// Convert nCurrGantry to um (smaller number) to read out in epics
M2L0.fCurrGantryY_um := LINT_TO_REAL(M2L0.nCurrGantryY) / 1000;
M2L0.fCurrGantryX_um := LINT_TO_REAL(M2L0.nCurrGantryX) / 1000;

// FB_MotionStage's for non-piezo axes
fbMotionStage_m7(stMotionStage:=M7);
fbMotionStage_m8(stMotionStage:=M8);
fbMotionStage_m9(stMotionStage:=M9);
fbMotionStage_m10(stMotionStage:=M10);
fbMotionStage_m11(stMotionStage:=M11);
fbMotionStage_m12(stMotionStage:=M12);

// Calculate RMS Error:
fbYRMSErrorM2L0(stMotionStage:=M7,
                fMaxRMSError=>fMaxYRMSErrorM2L0,
                fMinRMSError=>fMinYRMSErrorM2L0);

fbXRMSErrorM2L0(stMotionStage:=M9,
                fMaxRMSError=>fMaxXRMSErrorM2L0,
                fMinRMSError=>fMinXRMSErrorM2L0);

fbPitchRMSErrorM2L0(stMotionStage:=M11,
                fMaxRMSError=>fMaxPitchRMSErrorM2L0,
                fMinRMSError=>fMinPitchRMSErrorM2L0);

fbBenderRMSErrorM2L0(stMotionStage:=M12,
                fMaxRMSError=>fMaxBenderRMSErrorM2L0,
                fMinRMSError=>fMinBenderRMSErrorM2L0);

// Pitch Control
//fbM2L0PitchControl(Pitch:=GVL_M2L0.M2L0_Pitch,
                   //Stepper:=M11,
                   //lrCurrentSetpoint:=M11.fPosition,
                   //q_bDone=>bM2L0PitchDone,
                   //q_bBusy=>bM2L0PitchBusy);
// When STO hit, need to reset SP
//IF NOT M11.bHardwareEnable THEN
    //M11.fPosition := M11.stAxisStatus.fActPosition;
//END_IF

// Raw Encoder Counts For Epics
nEncCntYupM2L0 := ULINT_TO_UDINT(M2L0.fbRunHOMS.stYupEnc.Count);
nEncCntYdwnM2L0 := ULINT_TO_UDINT(M2L0.fbRunHOMS.stYdwnEnc.Count);
nEncCntXupM2L0 := ULINT_TO_UDINT(M2L0.fbRunHOMS.stXupEnc.Count);
nEncCntXdwnM2L0 := ULINT_TO_UDINT(M2L0.fbRunHOMS.stXdwnEnc.Count);
nEncCntPitchM2L0 := LINT_TO_UDINT(GVL_M2L0.M2L0_Pitch.diEncCnt);

// Encoder Reference Values For Epics
nEncRefYupM2L0 := ULINT_TO_UDINT(GVL_M2L0_Constants.nYUP_ENC_REF);
nEncRefYdwnM2L0 := ULINT_TO_UDINT(GVL_M2L0_Constants.nYDWN_ENC_REF);
nEncRefXupM2L0 := ULINT_TO_UDINT(GVL_M2L0_Constants.nXUP_ENC_REF);
nEncRefXdwnM2L0 := ULINT_TO_UDINT(GVL_M2L0_Constants.nXDWN_ENC_REF);
mcReadParameterPitchM2L0(Axis:=M11.Axis,
                         Enable:=TRUE,
                         ParameterNumber:=MC_AxisParameter.AxisEncoderOffset,
                         ReadMode:=READMODE_CYCLIC,
                         Value=>fEncRefPitchM2L0_urad);

nEncRefPitchM2L0 := LREAL_TO_UDINT(ABS(fEncRefPitchM2L0_urad) * fEncLeverArm_mm);

//Coatings States With PMPS
M7.bPowerSelf :=FALSE;


//SP1L0

// FB_MotionStage's for non-piezo axes
fbMotionStage_m13(stMotionStage:=M13);
fbMotionStage_m14(stMotionStage:=M14);
fbMotionStage_m15(stMotionStage:=M15);
fbMotionStage_m16(stMotionStage:=M16);
fbMotionStage_m17(stMotionStage:=M17);


M13.bHardwareEnable := bSTO AND bTH1_POTL AND bTH1_NOTL;
M14.bHardwareEnable := bSTO AND bTH2_POTL AND bTH2_NOTL;
M15.bHardwareEnable := bSTO AND bTX_POTL AND bTX_NOTL;
M16.bHardwareEnable := bSTO;
M17.bHardwareEnable := bSTO;


    //Turn on Fan by default
    bFanOn := TRUE;






P_CoatingProtections();


// Logging
fbLogHandler();

END_PROGRAM

// ---- POUs/P_CoatingProtections.TcPOU
PROGRAM P_CoatingProtections
VAR
        fbStripProtMR1L0 : FB_MirrorTwoCoatingProtection := (
            sDevName := 'MR1L0:HOMS',
            nUpperCoatingBoundary := 13300000,
            sUpperCoatingType := 'L0-B4C',
            nLowerCoatingBoundary := 11800000,
            sLowerCoatingType := 'L0-NICKEL');

        fbStripProtMR2L0 : FB_MirrorTwoCoatingProtection := (
            sDevName := 'MR2L0:HOMS',
            nUpperCoatingBoundary := 14300000,
            sUpperCoatingType := 'NICKEL',
            nLowerCoatingBoundary := 12800000,
            sLowerCoatingType := 'B4C');
END_VAR

fbStripProtMR1L0(
    FFO := GVL_PMPS.g_FastFaultOutput1,
    nCurrentEncoderCount := MAIN.nEncCntYupM1L0,
    neVRange := PMPS.PMPS_GVL.stCurrentBeamParameters.neVRange,
    bReadPmpsDb:= MOTION_GVL.fbStandardPMPSDB.bReadPmpsDb,
    bUsePmpsDb := TRUE,
   );

fbStripProtMR2L0(
    FFO := GVL_PMPS.g_FastFaultOutput1,
    nCurrentEncoderCount := MAIN.nEncCntYupM2L0,
    neVRange := PMPS.PMPS_GVL.stCurrentBeamParameters.neVRange,
    bReadPmpsDb:= MOTION_GVL.fbStandardPMPSDB.bReadPmpsDb,
    bUsePmpsDb := TRUE,
);

END_PROGRAM

// ---- POUs/PRG_1_PlcTask.TcPOU
PROGRAM PRG_1_PlcTask
VAR

END_VAR

PRG_MR1L0_HOMS();
PRG_MR2L0_HOMS();
PRG_SP1L0_DCCM();
PRG_PMPS();

END_PROGRAM

// ---- POUs/PRG_MR1L0_HOMS.TcPOU
PROGRAM PRG_MR1L0_HOMS
VAR
    {attribute 'pytmc' := 'pv: MR1L0:HOMS:COATING'}
    fbCoatingStates: FB_PositionStatePMPS2D;
    {attribute 'pytmc' := '
      pv: MR1L0:HOMS:COATING:STATE:SET
      io: io
    '}
    eStateSet: E_MR1L0_CoatingStates;
    {attribute 'pytmc' := '
      pv: MR1L0:HOMS:COATING:STATE:GET
      io: i
    '}
    eStateGet: E_MR1L0_CoatingStates;

    fbYSetup: FB_StateSetupHelper;

    fbPitchSetup: FB_StateSetupHelper;
    stDefaultPitch : ST_PositionState := (
        fDelta:=194.94,
        fVelocity:=100,
        fAccel:=390,
        fDecel:=390,
        bMoveOk:=TRUE,
        bValid:=TRUE,
        bUseRawCounts:=TRUE
    );
    astCoatingStatesY: ARRAY[1..GeneralConstants.MAX_STATES] OF ST_PositionState;
    astCoatingStatesPitch: ARRAY[1..GeneralConstants.MAX_STATES] OF ST_PositionState;

        // MR1L0 Flow Press Sensors
    {attribute 'TcLinkTo' := '.fbFlow_1.iRaw := TIIB[EL3054_M1L0_FWM_PRSM]^AI Standard Channel 1^Value;
                                 .fbFlow_2.iRaw := TIIB[EL3054_M1L0_FWM_PRSM]^AI Standard Channel 2^Value;
                              .fbPress_1.iRaw := TIIB[EL3054_M1L0_FWM_PRSM]^AI Standard Channel 3^Value
    '}
    {attribute 'pytmc' := '
        pv: MR1L0:HOMS
    '}
    fbCoolingPanel : FB_Axilon_Cooling_2f1p;
    {attribute 'TcLinkTo' := 'TIIB[EP2008-0001_M1M2_VCV]^Channel 1^Output'}
    {attribute 'pytmc' := '
        pv: MR1L0:HOMS:VCV
        io: io
        field: ZNAM OFF
        field: ONAM ON
    '}
    bActivateVarCoolMR1L0 AT %Q* : BOOL;
END_VAR

fbYSetup(stPositionState:=GVL_States.stDefaultY, bSetDefault:=TRUE);
fbPitchSetup(stPositionState:=stDefaultPitch, bSetDefault:=TRUE);

// MR1L0 B4C
fbYSetup(stPositionState:=astCoatingStatesY[E_MR1L0_CoatingStates.L0B4C],
    sName:='L0B4C',
    sPmpsState:='MR1L0:HOMS-L0-B4C',
    nEncoderCount:=21171800
);
fbPitchSetup(stPositionState:=astCoatingStatesPitch[E_MR1L0_CoatingStates.L0B4C],
    sName:='L0B4C',
    sPmpsState:='MR1L0:HOMS-L0-B4C',
    nEncoderCount:=8602330
);

// MR1L0 Ni
fbYSetup(stPositionState:=astCoatingStatesY[E_MR1L0_CoatingStates.L0Ni],
    sName:='L0Ni',
    sPmpsState:='MR1L0:HOMS-L0-NICKEL',
    nEncoderCount:=9171800
);
fbPitchSetup(stPositionState:=astCoatingStatesPitch[E_MR1L0_CoatingStates.L0Ni],
    sName:='L0Ni',
    sPmpsState:='MR1L0:HOMS-L0-NICKEL',
    nEncoderCount:=8602330
);

// MR1L0_L1 B4C
fbYSetup(stPositionState:=astCoatingStatesY[E_MR1L0_CoatingStates.L1B4C],
    bValid:=FALSE,
    sName:='L1B4C',
    sPmpsState:='MR1L0:HOMS-L1-B4C',
    nEncoderCount:=21171800
);
fbPitchSetup(stPositionState:=astCoatingStatesPitch[E_MR1L0_CoatingStates.L1B4C],
    bValid:=FALSE,
    sName:='L1B4C',
    sPmpsState:='MR1L0:HOMS-L1-B4C',
    nEncoderCount:=11116030,
    fDelta:=974.66
);

// MR1L0_L1 Ni
fbYSetup(stPositionState:=astCoatingStatesY[E_MR1L0_CoatingStates.L1Ni],
    bValid:=FALSE,
    sName:='L1Ni',
    sPmpsState:='MR1L0:HOMS-L1-NICKEL',
    nEncoderCount:=9171800
);
fbPitchSetup(stPositionState:=astCoatingStatesPitch[E_MR1L0_CoatingStates.L1Ni],
    bValid:=FALSE,
    sName:='L1Ni',
    sPmpsState:='MR1L0:HOMS-L1-NICKEL',
    nEncoderCount:=11116030,
    fDelta:=974.66
);

fbCoatingStates(
    stMotionStage1:=Main.M1,
    stMotionStage2:=Main.M5,
    astPositionState1:=astCoatingStatesY,
    astPositionState2:=astCoatingStatesPitch,
    eEnumSet:=eStateSet,
    eEnumGet:=eStateGet,
    fbFFHWO:=GVL_PMPS.g_FastFaultOutput1,
    fbArbiter:=GVL_PMPS.g_fbArbiter1,
    bEnableMotion:=TRUE,
    bEnableBeamParams:=TRUE,
    sDeviceName:='MR1L0:HOMS',
    sTransitionKey:='MR1L0:HOMS-TRANSITION',
);

fbCoolingPanel();

END_PROGRAM

// ---- POUs/PRG_MR2L0_HOMS.TcPOU
PROGRAM PRG_MR2L0_HOMS
VAR
    {attribute 'pytmc' := 'pv: MR2L0:HOMS:COATING'}
    fbCoatingStates: FB_PositionStatePMPS1D;
    {attribute 'pytmc' := '
      pv: MR2L0:HOMS:COATING:STATE:SET
      io: io
    '}
    eStateSet: E_MR2L0_CoatingStates;
    {attribute 'pytmc' := '
      pv: MR2L0:HOMS:COATING:STATE:GET
      io: i
    '}
    eStateGet: E_MR2L0_CoatingStates;
    fbYSetup: FB_StateSetupHelper;
    astCoatingStatesY: ARRAY[1..GeneralConstants.MAX_STATES] OF ST_PositionState;

    // MR2L0 Flow Press Sensors
    {attribute 'TcLinkTo' := '.fbFlow_1.iRaw := TIIB[EL3054_M2L0_FWM_PRSM]^AI Standard Channel 1^Value;
                                 .fbFlow_2.iRaw := TIIB[EL3054_M2L0_FWM_PRSM]^AI Standard Channel 2^Value;
                              .fbPress_1.iRaw := TIIB[EL3054_M2L0_FWM_PRSM]^AI Standard Channel 3^Value
    '}
    {attribute 'pytmc' := '
        pv: MR2L0:HOMS
    '}
    fbCoolingPanel : FB_Axilon_Cooling_2f1p;
        {attribute 'TcLinkTo' := 'TIIB[EP2008-0001_M1M2_VCV]^Channel 2^Output'}
    {attribute 'pytmc' := '
        pv: MR2L0:HOMS:VCV
        io: io
        field: ZNAM OFF
        field: ONAM ON
    '}
    bActivateVarCoolMR2L0 AT %Q* : BOOL;

END_VAR

fbYSetup(stPositionState:=GVL_States.stDefaultY, bSetDefault:=TRUE);

// MR2L0 B4C
fbYSetup(stPositionState:=astCoatingStatesY[E_MR2L0_CoatingStates.B4C],
    sName:='B4C',
    sPmpsState:='MR2L0:HOMS-B4C',
    nEncoderCount:=7018200
);

// MR2L0 Ni
fbYSetup(stPositionState:=astCoatingStatesY[E_MR2L0_CoatingStates.Ni],
    sName:='Ni',
    sPmpsState:='MR2L0:HOMS-NICKEL',
    nEncoderCount:= 16018200
);

fbCoatingStates(
    stMotionStage:=Main.M7,
    astPositionState:=astCoatingStatesY,
    eEnumSet:=eStateSet,
    eEnumGet:=eStateGet,
    fbFFHWO:=GVL_PMPS.g_FastFaultOutput1,
    fbArbiter:=GVL_PMPS.g_fbArbiter1,
    bEnableMotion:=TRUE,
    bEnableBeamParams:=TRUE,
    sDeviceName:='MR2L0:HOMS',
    sTransitionKey:='MR2L0:HOMS-TRANSITION',
);

fbCoolingPanel();

END_PROGRAM

// ---- POUs/PRG_SP1L0_DCCM.TcPOU
PROGRAM PRG_SP1L0_DCCM
VAR

END_VAR

END_PROGRAM

// ---- POUs/PRG_PMPS.TcPOU
PROGRAM PRG_PMPS
VAR
    // PMPS arbiter interface
    fbArbiterIO : FB_SubSysToArbiter_IO;
    {attribute 'TcLinkTo' := 'TIIB[PMPS_PRE]^IO Outputs^MR1L0_Pitch_ENC'}
    nMR1L0_Pitch_ENC_PMPS AT %Q* : ULINT;

END_VAR

// PMPS
MOTION_GVL.fbStandardPMPSDB(
    io_fbFFHWO:=GVL_PMPS.g_FastFaultOutput1,
    bEnable:=TRUE,
    sPLCName:='plc-lfe-optics'
);

GVL_PMPS.g_fbArbiter1.AddRequest(16#5, PMPS_GVL.cstFullBeam, 'LFE Optics');
fbArbiterIO(Arbiter := GVL_PMPS.g_fbArbiter1, fbFFHWO := GVL_PMPS.g_FastFaultOutput1);
GVL_PMPS.g_FastFaultOutput1.Execute(i_xVeto:=);
GVL_PMPS.g_FastFaultOutput2.Execute(i_xVeto:=);

 nMR1L0_Pitch_ENC_PMPS := Main.M5.nRawEncoderULINT;

END_PROGRAM

// ---- POUs/Serial Comm/P_Serial_Com.TcPOU
PROGRAM P_Serial_Com
VAR
    fbSerialLineControl_EL6001_M1L0: SerialLineControl; // M1L0 Serial Comm Function Block
    fbSerialLineControl_EL6001_M2L0: SerialLineControl; // M2L0 Serial Comm Function Block
END_VAR

// These are the global IOs...don't forget to copy your data into them

(* EL6001 Serial port 0 com function *)
fbSerialLineControl_EL6001_M1L0(Mode:= SERIALLINEMODE_EL6_22B,
                                pComIn:= ADR(Serial_stComIn_M1L0),
                                   pComOut:=ADR(Serial_stComOut_M1L0),
                                SizeComIn:= SIZEOF(Serial_stComIn_M1L0),
                                TxBuffer:= Serial_TXBuffer_M1L0,
                                RxBuffer:= Serial_RXBuffer_M1L0,
                                Error=>,
                                ErrorID=>);

fbSerialLineControl_EL6001_M2L0(Mode:= SERIALLINEMODE_EL6_22B,
                                pComIn:= ADR(Serial_stComIn_M2L0),
                                   pComOut:=ADR(Serial_stComOut_M2L0),
                                SizeComIn:= SIZEOF(Serial_stComIn_M2L0),
                                TxBuffer:= Serial_TXBuffer_M2L0,
                                RxBuffer:= Serial_RXBuffer_M2L0,
                                Error=>,
                                ErrorID=>);

END_PROGRAM
